// Mitsubishi GX Works2 project: barier_control   PLC: FX1N/FX1NC

PROGRAM MAIN
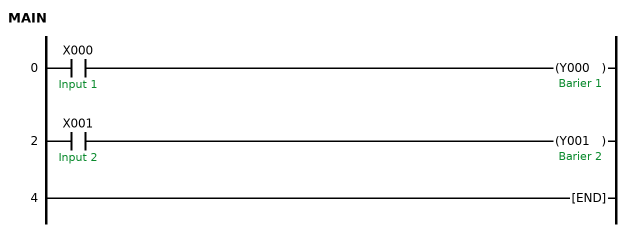
0     LD      X000  ; Input 1
      OUT     Y000  ; Barier 1
2     LD      X001  ; Input 2
      OUT     Y001  ; Barier 2
4     END
END_PROGRAM
